PROGRAM MAIN
VAR
END_VAR


// PLC Methode
 HmiMapping();
 HmiFunctionAddition();
 HmiFunctionLizenz();

// Hmi Classic

// Hmi Vue3

// Testing

END_PROGRAM

(* stored: Version 1.1.0.1, ProductVersion 3.1.4024.12
   POU MAIN: Id {6229951d-7c2a-451d-aeaf-626ebb47240f}, SpecialFunc None *)
